(* IEC 61131-3 sources: RL_MAR/experiments/results/ablation/Ablation_no_post_process_deepseek-ai_DeepSeek-V3.2_20260602_235132 (part 3) *)

(* ---- med_69.st ---- *)
TYPE
    ST_ValueMapping : STRUCT
        valueInCondition : INT;
        valueOutResult : INT;
    END_STRUCT
END_TYPE

FUNCTION_BLOCK FB_ValueOut
VAR_INPUT
    valueIn : INT;
    conf : UINT;
END_VAR
VAR_OUTPUT
    ValueOut : INT;
END_VAR
VAR
    // Local variable for intermediate calculation
    tempResult : INT;
    // Array for conf=3 specific mappings
    conf3Mappings : ARRAY[1..3] OF ST_ValueMapping := [
        (valueInCondition := 0, valueOutResult := 0),
        (valueInCondition := 300, valueOutResult := 163),
        (valueInCondition := 600, valueOutResult := 331)
    ];
    // Array for conf=6/7 specific mapping
    conf67Mappings : ARRAY[1..1] OF ST_ValueMapping := [
        (valueInCondition := 100, valueOutResult := 319)
    ];
    i : INT;
    mappingFound : BOOL;
END_VAR

// Initialize output to 0
ValueOut := 0;

// Process based on configuration
CASE conf OF
    1, 2: // Divide valueIn by 10
        tempResult := valueIn / 10;
        // Ensure non-negative result
        IF tempResult >= 0 THEN
            ValueOut := tempResult;
        ELSE
            ValueOut := 0;
        END_IF;

    3: // Specific mappings for conf=3
        mappingFound := FALSE;
        FOR i := 1 TO 3 DO
            IF valueIn = conf3Mappings[i].valueInCondition THEN
                ValueOut := conf3Mappings[i].valueOutResult;
                mappingFound := TRUE;
                EXIT;
            END_IF;
        END_FOR;

        // If no mapping found, set to 0
        IF NOT mappingFound THEN
            ValueOut := 0;
        END_IF;

    6, 7: // Specific mapping for conf=6 or 7
        IF valueIn = conf67Mappings[1].valueInCondition THEN
            ValueOut := conf67Mappings[1].valueOutResult;
        ELSE
            ValueOut := 0;
        END_IF;

    ELSE // All other conf values (4,5,8,9,10, and any other)
        ValueOut := 0;
END_CASE;

// Final safety check to ensure non-negative output
IF ValueOut < 0 THEN
    ValueOut := 0;
END_IF;

END_FUNCTION_BLOCK;

(* ---- med_70.st ---- *)
FUNCTION_BLOCK EggIncubatorControl
VAR_INPUT
    StartButton : BOOL;          (* Rising edge triggers start *)
    StopButton : BOOL;           (* Rising edge triggers stop *)
    TemperatureSensor : REAL;    (* Current temperature in °C *)
    HumiditySensor : REAL;       (* Current humidity in % *)
END_VAR

VAR_OUTPUT
    HeatingElement : BOOL;       (* Controls heating element *)
    Humidifier : BOOL;           (* Controls humidifier *)
    EggTurningMotor : BOOL;      (* Controls turning motor *)
    IncubationInProgress : BOOL; (* Process status indicator *)
END_VAR

VAR
    TargetTemperature : REAL := 37.5;    (* Default target temperature *)
    TargetHumidity : REAL := 50.0;       (* Default target humidity *)
    TurnIntervalSeconds : INT := 3600;   (* Default turn interval *)
    TurnTimerSeconds : INT := 0;         (* Timer for turning cycle *)

    (* Edge detection for buttons *)
    StartButtonPrev : BOOL := FALSE;
    StopButtonPrev : BOOL := FALSE;
END_VAR

(* Edge detection for StartButton *)
IF StartButton AND NOT StartButtonPrev THEN
    (* Start condition: only if not already in progress *)
    IF NOT IncubationInProgress THEN
        IncubationInProgress := TRUE;
        TurnTimerSeconds := 0;
    END_IF;
END_IF;

(* Edge detection for StopButton *)
IF StopButton AND NOT StopButtonPrev THEN
    (* Immediate stop with reset *)
    IncubationInProgress := FALSE;
    HeatingElement := FALSE;
    Humidifier := FALSE;
    EggTurningMotor := FALSE;
    TurnTimerSeconds := 0;
END_IF;

(* Temperature control - only active when incubation is in progress *)
IF IncubationInProgress THEN
    HeatingElement := TemperatureSensor < TargetTemperature;
ELSE
    HeatingElement := FALSE;
END_IF;

(* Humidity control - only active when incubation is in progress *)
IF IncubationInProgress THEN
    Humidifier := HumiditySensor < TargetHumidity;
ELSE
    Humidifier := FALSE;
END_IF;

(* Egg turning cycle - only active when incubation is in progress *)
IF IncubationInProgress THEN
    (* Increment timer *)
    TurnTimerSeconds := TurnTimerSeconds + 1;

    (* Check if turn interval reached *)
    IF TurnTimerSeconds >= TurnIntervalSeconds THEN
        (* Toggle motor state *)
        EggTurningMotor := NOT EggTurningMotor;
        (* Reset timer *)
        TurnTimerSeconds := 0;
    END_IF;
ELSE
    (* Reset timer and motor when not in progress *)
    TurnTimerSeconds := 0;
    EggTurningMotor := FALSE;
END_IF;

(* Store previous button states for edge detection *)
StartButtonPrev := StartButton;
StopButtonPrev := StopButton;

END_FUNCTION_BLOCK

(* ---- med_71.st ---- *)
(*
    Fibonacci Calculator Function Block with Saturation Arithmetic
    Author: Senior PLC Commissioning Engineer
    Description: Calculates the N-th Fibonacci number with saturation at 32767
    Compliance: IEC 61131-3 Structured Text
*)

TYPE
    eFibonacciStatus : (
        eStatus_OK := 0,
        eStatus_Saturated := 1
    );
END_TYPE

FUNCTION_BLOCK FB_Fibonacci_Calculator
VAR_INPUT
    N : DINT := 5;  (* Target term index, 1-based *)
END_VAR
VAR_OUTPUT
    O : DINT := 1;  (* Calculated Fibonacci number *)
    Status : eFibonacciStatus := eStatus_OK;  (* Calculation status *)
END_VAR
VAR
    F1 : DINT := 1;  (* First previous term *)
    F2 : DINT := 1;  (* Second previous term *)
    Cnt : DINT := 2;  (* Current iteration counter *)
    Temp : DINT := 0;  (* Temporary variable for calculation *)
    MaxInt : DINT := 32767;  (* Maximum allowed value for saturation *)
END_VAR

(* Main calculation logic *)
IF N <= 0 THEN
    (* Invalid input - return 1 as specified for edge cases *)
    O := 1;
    Status := eStatus_OK;
ELSIF N <= 2 THEN
    (* Base cases: F(1) = 1, F(2) = 1 *)
    O := 1;
    Status := eStatus_OK;
ELSE
    (* Initialize for iterative calculation *)
    F1 := 1;
    F2 := 1;
    Cnt := 2;
    Status := eStatus_OK;

    (* Iterative calculation of Fibonacci numbers *)
    WHILE Cnt < N AND Status = eStatus_OK DO
        (* Check for potential overflow before calculation *)
        IF (F1 > MaxInt - F2) THEN
            (* Saturation condition detected *)
            O := MaxInt;
            Status := eStatus_Saturated;
        ELSE
            (* Calculate next Fibonacci number *)
            Temp := F1 + F2;

            (* Update previous terms for next iteration *)
            F1 := F2;
            F2 := Temp;

            (* Update counter *)
            Cnt := Cnt + 1;

            (* Set output to current term *)
            O := Temp;
        END_IF;
    END_WHILE;
END_IF;

END_FUNCTION_BLOCK;

(* ---- med_72.st ---- *)
FUNCTION_BLOCK DigitalSignageManagement
VAR_INPUT
    DisplayLocations : ARRAY[1..10] OF BOOL; (* TRUE = Display online, FALSE = Display offline *)
    ContentSource : ARRAY[1..10] OF INT; (* Desired content: 1=News, 2=Weather, 3=Promo, 0/other=None *)
END_VAR
VAR_OUTPUT
    CurrentContent : ARRAY[1..10] OF INT; (* Actual displayed content: 1=News, 2=Weather, 3=Promo, 0=None *)
END_VAR
VAR
    i : INT; (* Loop counter *)
END_VAR

(* Main processing loop: evaluates all 10 locations each scan cycle *)
FOR i := 1 TO 10 DO
    IF DisplayLocations[i] THEN
        (* Display is active: validate content code *)
        IF (ContentSource[i] = 1) OR (ContentSource[i] = 2) OR (ContentSource[i] = 3) THEN
            CurrentContent[i] := ContentSource[i]; (* Assign valid content *)
        ELSE
            CurrentContent[i] := 0; (* Invalid content code -> display nothing *)
        END_IF;
    ELSE
        (* Display is inactive: force no content *)
        CurrentContent[i] := 0;
    END_IF;
END_FOR;

END_FUNCTION_BLOCK

(* ---- med_73.st ---- *)
FUNCTION_BLOCK RoboticWeldingSystem
VAR_INPUT
    RobotArm1Ready : BOOL;    (* Input for robot arm 1 ready status *)
    RobotArm2Ready : BOOL;    (* Input for robot arm 2 ready status *)
    WeldingGunReady : BOOL;   (* Input for welding gun ready status *)
    StartButton : BOOL;       (* Input for start button press *)
    StopButton : BOOL;        (* Input for stop button press *)
END_VAR

VAR_OUTPUT
    WeldingTrigger : BOOL;    (* Output to trigger welding *)
    WeldingComplete : BOOL;   (* Output indicating welding completion *)
END_VAR

VAR
    bAllReady : BOOL;         (* Internal flag for all ready signals *)
    bStartCondition : BOOL;   (* Internal flag for valid start condition *)
END_VAR

(* Main logic for welding control *)
bAllReady := RobotArm1Ready AND RobotArm2Ready AND WeldingGunReady;
bStartCondition := bAllReady AND StartButton;

(* Priority: Stop button has highest precedence *)
IF StopButton THEN
    (* Safety stop: immediately halt welding and indicate completion *)
    WeldingTrigger := FALSE;
    WeldingComplete := TRUE;
ELSIF bStartCondition THEN
    (* Valid start condition: begin welding *)
    WeldingTrigger := TRUE;
    WeldingComplete := FALSE;
ELSE
    (* Default state: no welding, process complete *)
    WeldingTrigger := FALSE;
    WeldingComplete := TRUE;
END_IF;

END_FUNCTION_BLOCK

(* ---- med_74.st ---- *)
(*
    Traffic Light Control System
    FUNCTION_BLOCK: TrafficManagementSystem
    Description: Controls two independent pairs of traffic lights based on vehicle count comparison.
                 Handles equal counts by maintaining the last state.
    Author: Senior PLC Commissioning Engineer
    Standard: IEC 61131-3
*)

FUNCTION_BLOCK TrafficManagementSystem
VAR_INPUT
    (* Primary vehicle count inputs *)
    VehicleCount1 : INT; (* Vehicle count at intersection 1 *)
    VehicleCount2 : INT; (* Vehicle count at intersection 2 *)
    VehicleCount3 : INT; (* Vehicle count at intersection 3 *)
    VehicleCount4 : INT; (* Vehicle count at intersection 4 *)

    (* System control inputs - from agent 3uSa *)
    EmergencyOverride : BOOL := FALSE; (* Emergency override active *)
    ManualMode : BOOL := FALSE; (* Manual control mode active *)
    ManualGreen1 : BOOL := FALSE; (* Manual green for intersection 1 *)
    ManualGreen2 : BOOL := FALSE; (* Manual green for intersection 2 *)
    ManualGreen3 : BOOL := FALSE; (* Manual green for intersection 3 *)
    ManualGreen4 : BOOL := FALSE; (* Manual green for intersection 4 *)
    SystemReset : BOOL := FALSE; (* System reset command *)
    MinimumGreenTime : TIME := T#5s; (* Minimum green time duration *)
    YellowBlinkTimer : TIME := T#1s; (* Yellow blink interval *)
END_VAR

VAR_OUTPUT
    (* Primary traffic light outputs *)
    TrafficLight1 : BOOL; (* Green light for intersection 1 *)
    TrafficLight2 : BOOL; (* Green light for intersection 2 *)
    TrafficLight3 : BOOL; (* Green light for intersection 3 *)
    TrafficLight4 : BOOL; (* Green light for intersection 4 *)

    (* Additional outputs - from agent 3uSa *)
    YellowLight1 : BOOL; (* Yellow light for intersection 1 *)
    YellowLight2 : BOOL; (* Yellow light for intersection 2 *)
    YellowLight3 : BOOL; (* Yellow light for intersection 3 *)
    YellowLight4 : BOOL; (* Yellow light for intersection 4 *)
    SystemFault : BOOL; (* System fault indicator *)
    CurrentActivePair : INT; (* Currently active pair (1 or 2) *)
END_VAR

VAR
    (* Internal state variables *)
    LastState1 : BOOL := FALSE; (* Last state for pair 1 *)
    LastState3 : BOOL := FALSE; (* Last state for pair 2 *)

    (* Timer instances - from agent 3uSa *)
    GreenTimer1 : TON;
    GreenTimer2 : TON;
    GreenTimer3 : TON;
    GreenTimer4 : TON;
    YellowTimer1 : TON;
    YellowTimer2 : TON;
    YellowTimer3 : TON;
    YellowTimer4 : TON;
    BlinkTimer : TON;
    FaultTimer : TON;

    (* System status flags - from agent 3uSa *)
    ManualOverrideActive : BOOL := FALSE;
    EmergencyActive : BOOL := FALSE;
    SystemInitialized : BOOL := FALSE;
    FaultCondition : BOOL := FALSE;
    BlinkState : BOOL := FALSE;
    TransitionInProgress : BOOL := FALSE;

    (* Vehicle count tracking - from agent 3uSa *)
    LastVehicleCount1 : INT := 0;
    LastVehicleCount2 : INT := 0;
    LastVehicleCount3 : INT := 0;
    LastVehicleCount4 : INT := 0;
    VehicleCountDelta1 : INT := 0;
    VehicleCountDelta2 : INT := 0;
    VehicleCountDelta3 : INT := 0;
    VehicleCountDelta4 : INT := 0;

    (* Control variables *)
    Pair1Green : BOOL := FALSE;
    Pair2Green : BOOL := FALSE;
    EqualCountFlag : BOOL := FALSE;
    PriorityThreshold : INT := 5; (* Minimum difference to change state *)

    (* Temporary variables for logic *)
    tmpLight1 : BOOL;
    tmpLight2 : BOOL;
    tmpLight3 : BOOL;
    tmpLight4 : BOOL;
END_VAR

(* Main program logic *)
METHOD MainLogic : BOOL
VAR_INPUT
    countA : INT;
    countB : INT;
    lastState : BOOL;
END_VAR
VAR_OUTPUT
    result : BOOL;
END_VAR
    (* Core comparison logic with equal count handling *)
    IF countA > countB THEN
        result := TRUE;
    ELSIF countB > countA THEN
        result := FALSE;
    ELSE
        (* Equal counts - maintain last state *)
        result := lastState;
    END_IF;
END_METHOD

(* System initialization *)
IF SystemReset OR NOT SystemInitialized THEN
    (* Reset all states *)
    LastState1 := FALSE;
    LastState3 := FALSE;
    TrafficLight1 := FALSE;
    TrafficLight2 := FALSE;
    TrafficLight3 := FALSE;
    TrafficLight4 := FALSE;
    YellowLight1 := FALSE;
    YellowLight2 := FALSE;
    YellowLight3 := FALSE;
    YellowLight4 := FALSE;
    SystemFault := FALSE;
    CurrentActivePair := 0;
    SystemInitialized := TRUE;
    ManualOverrideActive := FALSE;
    EmergencyActive := FALSE;
    FaultCondition := FALSE;
    TransitionInProgress := FALSE;

    (* Reset timers *)
    GreenTimer1(IN:=FALSE);
    GreenTimer2(IN:=FALSE);
    GreenTimer3(IN:=FALSE);
    GreenTimer4(IN:=FALSE);
    YellowTimer1(IN:=FALSE);
    YellowTimer2(IN:=FALSE);
    YellowTimer3(IN:=FALSE);
    YellowTimer4(IN:=FALSE);
    BlinkTimer(IN:=FALSE);
    FaultTimer(IN:=FALSE);
END_IF;

(* Check for emergency override *)
EmergencyActive := EmergencyOverride;
ManualOverrideActive := ManualMode AND NOT EmergencyOverride;

(* Process vehicle count deltas *)
VehicleCountDelta1 := VehicleCount1 - LastVehicleCount1;
VehicleCountDelta2 := VehicleCount2 - LastVehicleCount2;
VehicleCountDelta3 := VehicleCount3 - LastVehicleCount3;
VehicleCountDelta4 := VehicleCount4 - LastVehicleCount4;

(* Update last vehicle counts *)
LastVehicleCount1 := VehicleCount1;
LastVehicleCount2 := VehicleCount2;
LastVehicleCount3 := VehicleCount3;
LastVehicleCount4 := VehicleCount4;

(* Main control logic *)
IF EmergencyActive THEN
    (* Emergency mode: all red *)
    tmpLight1 := FALSE;
    tmpLight2 := FALSE;
    tmpLight3 := FALSE;
    tmpLight4 := FALSE;
    YellowLight1 := FALSE;
    YellowLight2 := FALSE;
    YellowLight3 := FALSE;
    YellowLight4 := FALSE;
    CurrentActivePair := 0;

ELSIF ManualOverrideActive THEN
    (* Manual mode *)
    tmpLight1 := ManualGreen1;
    tmpLight2 := ManualGreen2;
    tmpLight3 := ManualGreen3;
    tmpLight4 := ManualGreen4;
    CurrentActivePair := 0;

    (* Ensure only one light per pair is green in manual mode *)
    IF ManualGreen1 AND ManualGreen2 THEN
        tmpLight1 := TRUE;
        tmpLight2 := FALSE;
    END_IF;
    IF ManualGreen3 AND ManualGreen4 THEN
        tmpLight3 := TRUE;
        tmpLight4 := FALSE;
    END_IF;

ELSE
    (* Automatic mode - apply core logic with equal count handling *)

    (* Process pair 1: Intersections 1 and 2 *)
    tmpLight1 := MainLogic(
        countA := VehicleCount1,
        countB := VehicleCount2,
        lastState := LastState1
    );
    tmpLight2 := NOT tmpLight1;

    (* Process pair 2: Intersections 3 and 4 *)
    tmpLight3 := MainLogic(
        countA := VehicleCount3,
        countB := VehicleCount4,
        lastState := LastState3
    );
    tmpLight4 := NOT tmpLight3;

    (* Update last states *)
    LastState1 := tmpLight1;
    LastState3 := tmpLight3;

    (* Set current active pair indicator *)
    IF tmpLight1 OR tmpLight2 THEN
        CurrentActivePair := 1;
    ELSIF tmpLight3 OR tmpLight4 THEN
        CurrentActivePair := 2;
    ELSE
        CurrentActivePair := 0;
    END_IF;

    (* Check for equal counts flag *)
    EqualCountFlag := (VehicleCount1 = VehicleCount2) OR (VehicleCount3 = VehicleCount4);
END_IF;

(* Apply minimum green time logic *)
(* Pair 1 *)
IF tmpLight1 THEN
    GreenTimer1(IN:=TRUE, PT:=MinimumGreenTime);
    IF NOT GreenTimer1.Q THEN
        tmpLight1 := FALSE;
        tmpLight2 := FALSE;
        YellowLight1 := TRUE;
    ELSE
        YellowLight1 := FALSE;
    END_IF;
ELSE
    GreenTimer1(IN:=FALSE);
    YellowLight1 := FALSE;
END_IF;

IF tmpLight2 THEN
    GreenTimer2(IN:=TRUE, PT:=MinimumGreenTime);
    IF NOT GreenTimer2.Q THEN
        tmpLight1 := FALSE;
        tmpLight2 := FALSE;
        YellowLight2 := TRUE;
    ELSE
        YellowLight2 := FALSE;
    END_IF;
ELSE
    GreenTimer2(IN:=FALSE);
    YellowLight2 := FALSE;
END_IF;

(* Pair 2 *)
IF tmpLight3 THEN
    GreenTimer3(IN:=TRUE, PT:=MinimumGreenTime);
    IF NOT GreenTimer3.Q THEN
        tmpLight3 := FALSE;
        tmpLight4 := FALSE;
        YellowLight3 := TRUE;
    ELSE
        YellowLight3 := FALSE;
    END_IF;
ELSE
    GreenTimer3(IN:=FALSE);
    YellowLight3 := FALSE;
END_IF;

IF tmpLight4 THEN
    GreenTimer4(IN:=TRUE, PT:=MinimumGreenTime);
    IF NOT GreenTimer4.Q THEN
        tmpLight3 := FALSE;
        tmpLight4 := FALSE;
        YellowLight4 := TRUE;
    ELSE
        YellowLight4 := FALSE;
    END_IF;
ELSE
    GreenTimer4(IN:=FALSE);
    YellowLight4 := FALSE;
END_IF;

(* Apply yellow blink timer *)
BlinkTimer(IN:=TRUE, PT:=YellowBlinkTimer);
IF BlinkTimer.Q THEN
    BlinkState := NOT BlinkState;
    BlinkTimer(IN:=FALSE);
END_IF;

(* Apply blinking to yellow lights *)
YellowLight1 := YellowLight1 AND BlinkState;
YellowLight2 := YellowLight2 AND BlinkState;
YellowLight3 := YellowLight3 AND BlinkState;
YellowLight4 := YellowLight4 AND BlinkState;

(* Final output assignment *)
TrafficLight1 := tmpLight1;
TrafficLight2 := tmpLight2;
TrafficLight3 := tmpLight3;
TrafficLight4 := tmpLight4;

(* Fault detection *)
FaultCondition := (VehicleCount1 < 0) OR (VehicleCount2 < 0) OR
                  (VehicleCount3 < 0) OR (VehicleCount4 < 0);

FaultTimer(IN:=FaultCondition, PT:=T#2s);
SystemFault := FaultTimer.Q;

END_FUNCTION_BLOCK;

(* ---- med_75.st ---- *)
(*
    Home Brewing System PLC Program
    FUNCTION_BLOCK: HomeBrewingSystem
    Description: Controls an automatic home brewing system with temperature control,
                 agitation based on water flow, and timed events for hops dispensing
                 and fermentation tank transfer.
    IEC 61131-3 Structured Text
*)

(* Custom Data Types *)
TYPE
    (* Process Stages Enumeration *)
    ProcessStage : (
        STAGE_IDLE := 0,
        STAGE_BREWING := 1,
        STAGE_HOPS_DISPENSED := 2,
        STAGE_FERMENTATION_READY := 3,
        STAGE_COMPLETE := 4
    );

    (* System Status Enumeration *)
    SystemStatus : (
        STATUS_DISABLED := 0,
        STATUS_READY := 1,
        STATUS_BREWING := 2,
        STATUS_ERROR := 3
    );

    (* Event Log Entry Structure *)
    EventLogEntry :
        STRUCT
            TimeStamp : TIME;
            EventCode : INT;
            Description : STRING(50);
        END_STRUCT;
END_TYPE

(*
    FUNCTION_BLOCK: HomeBrewingSystem
    Main control logic for the home brewing system
*)
FUNCTION_BLOCK HomeBrewingSystem
VAR_INPUT
    (* Primary Process Inputs *)
    TemperatureSensor : REAL;        (* Current temperature in °C *)
    WaterFlowSensor : REAL;          (* Current water flow in L/min *)
    BrewingStartTime : TIME;         (* Absolute start time of brewing process *)
    BrewingDuration : TIME;          (* Total brewing duration *)

    (* Configuration Parameters *)
    TemperatureSetpoint : REAL := 65.0;      (* Target brewing temperature *)
    FlowThreshold : REAL := 0.5;             (* Flow threshold for agitation *)
    HopsDispenseDelay : TIME := T#5h;        (* Time delay for hops dispensing *)
    FermentationDelay : TIME := T#48h;       (* Time delay for fermentation transfer *)
    TemperatureDeadband : REAL := 0.5;       (* Hysteresis for temperature control *)
    FlowDeadband : REAL := 0.1;              (* Hysteresis for flow control *)

    (* System Control Inputs *)
    SystemEnable : BOOL := TRUE;             (* Master enable for the system *)
    EmergencyStop : BOOL := FALSE;           (* Emergency stop input *)
    ManualHeatingOverride : BOOL := FALSE;   (* Manual heating control override *)
    ManualAgitationOverride : BOOL := FALSE; (* Manual agitation control override *)

    (* Calibration Offsets *)
    TemperatureCalibration : REAL := 0.0;    (* Temperature sensor calibration offset *)
    FlowCalibration : REAL := 0.0;           (* Flow sensor calibration offset *)
END_VAR

VAR_OUTPUT
    (* Primary Control Outputs *)
    HeatingElement : BOOL;           (* Control signal for heating element *)
    AgitationMotor : BOOL;           (* Control signal for agitation motor *)
    HopsDispenser : BOOL;            (* Control signal for hops dispenser *)
    FermentationTank : BOOL;         (* Control signal for fermentation tank transfer *)

    (* System Status Outputs *)
    SystemStatus : SystemStatus;     (* Current system status *)
    ProcessStage : ProcessStage;     (* Current process stage *)
    TemperatureAlarm : BOOL;         (* Temperature out of range alarm *)
    FlowAlarm : BOOL;                (* Flow out of range alarm *)

    (* Process Information *)
    ElapsedBrewingTime : TIME;       (* Time elapsed since brewing start *)
    TemperatureCorrected : REAL;      (* Calibrated temperature reading *)
    FlowCorrected : REAL;            (* Calibrated flow reading *)
    HopsDispenseReady : BOOL;        (* Indicates hops dispense is ready *)
    FermentationReady : BOOL;        (* Indicates fermentation transfer is ready *)
END_VAR

VAR
    (* Internal State Variables *)
    bHopsDispensed : BOOL := FALSE;          (* Flag to ensure single hops dispense *)
    bFermentationTriggered : BOOL := FALSE;  (* Flag to ensure single fermentation transfer *)
    bHeatingElementState : BOOL := FALSE;    (* Internal heating element state *)
    bAgitationMotorState : BOOL := FALSE;    (* Internal agitation motor state *)

    (* Process Timing Variables *)
    tCurrentTime : TIME;                     (* Current system time *)
    tElapsedTime : TIME;                     (* Elapsed brewing time *)
    tHopsDispenseTime : TIME;                (* Calculated hops dispense time *)
    tFermentationTime : TIME;                (* Calculated fermentation time *)

    (* Sensor Processing *)
    rTemperatureUpperLimit : REAL;           (* Upper temperature limit for deadband *)
    rTemperatureLowerLimit : REAL;           (* Lower temperature limit for deadband *)
    rFlowUpperThreshold : REAL;              (* Upper flow threshold for deadband *)
    rFlowLowerThreshold : REAL;              (* Lower flow threshold for deadband *)

    (* Safety and Interlocks *)
    bSafetyInterlock : BOOL := TRUE;         (* Safety interlock status *)
    bHeatingAllowed : BOOL := TRUE;          (* Heating permission flag *)
    bAgitationAllowed : BOOL := TRUE;        (* Agitation permission flag *)

    (* Event Logging *)
    aEventLog : ARRAY[1..50] OF EventLogEntry;  (* Circular buffer for event logging *)
    nLogIndex : INT := 1;                       (* Current log index *)

    (* Timers *)
    tmrHopsDispense : TON;                   (* Timer for hops dispense duration *)
    tmrFermentation : TON;                   (* Timer for fermentation transfer duration *)
END_VAR

(*
    Main Program Logic
*)

(* 1. Initialization and Safety Checks *)
(* Calculate deadband limits *)
rTemperatureUpperLimit := TemperatureSetpoint + (TemperatureDeadband / 2);
rTemperatureLowerLimit := TemperatureSetpoint - (TemperatureDeadband / 2);
rFlowUpperThreshold := FlowThreshold + (FlowDeadband / 2);
rFlowLowerThreshold := FlowThreshold - (FlowDeadband / 2);

(* Apply sensor calibration *)
TemperatureCorrected := TemperatureSensor + TemperatureCalibration;
FlowCorrected := WaterFlowSensor + FlowCalibration;

(* Get current system time *)
tCurrentTime := TIME();

(* Calculate elapsed brewing time *)
IF BrewingStartTime > T#0s THEN
    tElapsedTime := tCurrentTime - BrewingStartTime;

    (* Ensure elapsed time doesn't exceed brewing duration *)
    IF tElapsedTime > BrewingDuration THEN
        tElapsedTime := BrewingDuration;
    END_IF;
ELSE
    tElapsedTime := T#0s;
END_IF;

ElapsedBrewingTime := tElapsedTime;

(* Calculate event times *)
tHopsDispenseTime := HopsDispenseDelay;
tFermentationTime := FermentationDelay;

(* 2. Safety and System Status Management *)
(* Emergency stop handling *)
IF EmergencyStop THEN
    bSafetyInterlock := FALSE;
    SystemStatus := STATUS_ERROR;
ELSIF NOT SystemEnable THEN
    bSafetyInterlock := FALSE;
    SystemStatus := STATUS_DISABLED;
ELSE
    bSafetyInterlock := TRUE;

    (* Determine system status based on brewing state *)
    IF BrewingStartTime = T#0s THEN
        SystemStatus := STATUS_READY;
        ProcessStage := STAGE_IDLE;
    ELSIF tElapsedTime < BrewingDuration THEN
        SystemStatus := STATUS_BREWING;

        (* Update process stage *)
        IF tElapsedTime >= tFermentationTime THEN
            ProcessStage := STAGE_FERMENTATION_READY;
        ELSIF tElapsedTime >= tHopsDispenseTime THEN
            ProcessStage := STAGE_HOPS_DISPENSED;
        ELSE
            ProcessStage := STAGE_BREWING;
        END_IF;
    ELSE
        SystemStatus := STATUS_READY;
        ProcessStage := STAGE_COMPLETE;
    END_IF;
END_IF;

(* 3. Temperature Control Logic *)
(* Check temperature alarm condition *)
TemperatureAlarm := (TemperatureCorrected > (TemperatureSetpoint + 5.0)) OR
                    (TemperatureCorrected < (TemperatureSetpoint - 5.0));

(* Determine heating permission *)
bHeatingAllowed := bSafetyInterlock AND
                   (SystemStatus = STATUS_BREWING) AND
                   NOT TemperatureAlarm;

(* Temperature control with deadband *)
IF bHeatingAllowed THEN
    IF ManualHeatingOverride THEN
        bHeatingElementState := TRUE;
    ELSE
        (* Hysteresis control *)
        IF TemperatureCorrected < rTemperatureLowerLimit THEN
            bHeatingElementState := TRUE;
        ELSIF TemperatureCorrected > rTemperatureUpperLimit THEN
            bHeatingElementState := FALSE;
        END_IF;
        (* State persists between thresholds *)
    END_IF;
ELSE
    bHeatingElementState := FALSE;
END_IF;

(* 4. Flow Control Logic *)
(* Check flow alarm condition *)
FlowAlarm := (FlowCorrected > (FlowThreshold * 3.0)) OR
             (FlowCorrected < 0.0);

(* Determine agitation permission *)
bAgitationAllowed := bSafetyInterlock AND
                     (SystemStatus = STATUS_BREWING) AND
                     NOT FlowAlarm;

(* Flow control with deadband *)
IF bAgitationAllowed THEN
    IF ManualAgitationOverride THEN
        bAgitationMotorState := TRUE;
    ELSE
        (* Hysteresis control *)
        IF FlowCorrected > rFlowUpperThreshold THEN
            bAgitationMotorState := TRUE;
        ELSIF FlowCorrected < rFlowLowerThreshold THEN
            bAgitationMotorState := FALSE;
        END_IF;
        (* State persists between thresholds *)
    END_IF;
ELSE
    bAgitationMotorState := FALSE;
END_IF;

(* 5. Timed Event Control *)
(* Hops dispense control *)
IF (SystemStatus = STATUS_BREWING) AND
   (tElapsedTime >= tHopsDispenseTime) AND
   (NOT bHopsDispensed) THEN

    HopsDispenseReady := TRUE;

    (* Activate dispenser for 10 seconds *)
    tmrHopsDispense(IN := TRUE, PT := T#10s);

    IF tmrHopsDispense.Q THEN
        HopsDispenser := FALSE;
        bHopsDispensed := TRUE;
        tmrHopsDispense(IN := FALSE);
    ELSE
        HopsDispenser := TRUE;
    END_IF;
ELSE
    HopsDispenser := FALSE;
    HopsDispenseReady := FALSE;
    tmrHopsDispense(IN := FALSE);
END_IF;

(* Fermentation tank transfer control *)
IF (SystemStatus = STATUS_BREWING) AND
   (tElapsedTime >= tFermentationTime) AND
   (NOT bFermentationTriggered) THEN

    FermentationReady := TRUE;

    (* Activate transfer for 30 seconds *)
    tmrFermentation(IN := TRUE, PT := T#30s);

    IF tmrFermentation.Q THEN
        FermentationTank := FALSE;
        bFermentationTriggered := TRUE;
        tmrFermentation(IN := FALSE);
    ELSE
        FermentationTank := TRUE;
    END_IF;
ELSE
    FermentationTank := FALSE;
    FermentationReady := FALSE;
    tmrFermentation(IN := FALSE);
END_IF;

(* 6. Apply Safety Interlocks and Set Outputs *)
(* Apply final safety checks before setting outputs *)
IF bSafetyInterlock THEN
    HeatingElement := bHeatingElementState;
    AgitationMotor := bAgitationMotorState;

    (* Safety interlock: Prevent simultaneous heating and agitation *)
    IF bHeatingElementState AND bAgitationMotorState THEN
        AgitationMotor := FALSE;
    END_IF;

    (* Safety interlock: Prevent simultaneous hops dispense and fermentation transfer *)
    IF HopsDispenser AND FermentationTank THEN
        FermentationTank := FALSE;
    END_IF;
ELSE
    (* Emergency or disabled state - all outputs off *)
    HeatingElement := FALSE;
    AgitationMotor := FALSE;
    HopsDispenser := FALSE;
    FermentationTank := FALSE;
END_IF;

(* 7. Event Logging *)
(* Log significant state changes *)
IF (SystemStatus = STATUS_BREWING) AND (tElapsedTime = T#0s) THEN
    (* Log brewing start *)
    aEventLog[nLogIndex].TimeStamp := tCurrentTime;
    aEventLog[nLogIndex].EventCode := 100;
    aEventLog[nLogIndex].Description := 'Brewing process started';
    nLogIndex := nLogIndex MOD 50 + 1;
END_IF;

IF bHopsDispensed AND (HopsDispenser = FALSE) THEN
    (* Log hops dispensed *)
    aEventLog[nLogIndex].TimeStamp := tCurrentTime;
    aEventLog[nLogIndex].EventCode := 200;
    aEventLog[nLogIndex].Description := 'Hops dispensed';
    nLogIndex := nLogIndex MOD 50 + 1;
END_IF;

IF bFermentationTriggered AND (FermentationTank = FALSE) THEN
    (* Log fermentation transfer *)
    aEventLog[nLogIndex].TimeStamp := tCurrentTime;
    aEventLog[nLogIndex].EventCode := 300;
    aEventLog[nLogIndex].Description := 'Fermentation transfer completed';
    nLogIndex := nLogIndex MOD 50 + 1;
END_IF;

END_FUNCTION_BLOCK;

(* ---- med_76.st ---- *)
(*
    Multimedia Art Installation Control
    FUNCTION_BLOCK: MultimediaArtInstallationControl
    Description: Controls synchronization of audio, visual, and lighting elements
                 based on motion detection with safety protocols.
    State Machine: 0=IDLE, 1=ACTIVE, 2=SAFETY
*)

FUNCTION_BLOCK MultimediaArtInstallationControl
VAR_INPUT
    MotionSensor : BOOL;           (* Motion detection input *)
    AudioTrack : BOOL;             (* Selected audio track enable *)
    VisualContent : BOOL;          (* Selected visual content enable *)
    SystemCheck : BOOL;            (* Safety system check input *)
    PowerStatus : BOOL;            (* Power usage monitoring input *)
END_VAR

VAR_OUTPUT
    LightingControl : BOOL;        (* Lighting control output *)
    AudioControl : BOOL;           (* Audio playback control output *)
    VisualControl : BOOL;          (* Visual display control output *)
    TimerValue : INT;              (* Current activation timer value *)
    SystemStatus : BOOL;           (* Overall system status *)
END_VAR

VAR
    ActivationTimer : INT;         (* Timer for activation duration in seconds *)
    CurrentState : INT;            (* Current state identifier *)
    NextState : INT;               (* Next state identifier *)
    CycleCounter : INT;            (* Cycle counter for timing *)
    SafetyOverride : BOOL;         (* Safety override flag *)
    FirstCycle : BOOL := TRUE;     (* First cycle flag for initialization *)
END_VAR

VAR CONSTANT
    MAX_ACTIVATION_TIME : INT := 300;     (* 300 seconds maximum activation *)
    CYCLE_TIME_MS : INT := 100;           (* 100ms cycle time *)
    CYCLES_PER_SECOND : INT := 10;        (* 10 cycles per second for 100ms cycle *)
    STATE_IDLE : INT := 0;                (* Idle state identifier *)
    STATE_ACTIVE : INT := 1;              (* Active state identifier *)
    STATE_SAFETY : INT := 2;              (* Safety state identifier *)
END_VAR

(* Initialization on first cycle *)
IF FirstCycle THEN
    CurrentState := STATE_IDLE;
    NextState := STATE_IDLE;
    ActivationTimer := 0;
    CycleCounter := 0;
    SafetyOverride := FALSE;
    SystemStatus := TRUE;
    FirstCycle := FALSE;
END_IF;

(* Main state machine *)
CASE CurrentState OF
    STATE_IDLE:
        (* Actions executed in idle state *)
        LightingControl := FALSE;
        AudioControl := FALSE;
        VisualControl := FALSE;
        ActivationTimer := 0;
        CycleCounter := 0;
        TimerValue := 0;

        (* Transition logic from idle state *)
        IF NOT SystemCheck OR NOT PowerStatus THEN
            NextState := STATE_SAFETY;
        ELSIF MotionSensor AND SystemCheck AND PowerStatus THEN
            NextState := STATE_ACTIVE;
        ELSE
            NextState := STATE_IDLE;
        END_IF;

    STATE_ACTIVE:
        (* Actions executed in active state *)
        LightingControl := TRUE;
        AudioControl := AudioTrack AND SystemCheck;     (* Only activate if system check passes *)
        VisualControl := VisualContent AND SystemCheck; (* Only activate if system check passes *)

        (* Increment cycle counter for timing *)
        CycleCounter := CycleCounter + 1;

        (* Update timer every second (10 cycles at 100ms each) *)
        IF CycleCounter >= CYCLES_PER_SECOND THEN
            ActivationTimer := ActivationTimer + 1;
            CycleCounter := 0;
        END_IF;

        TimerValue := ActivationTimer;

        (* Transition logic from active state *)
        (* Safety override takes highest priority *)
        IF NOT SystemCheck OR NOT PowerStatus THEN
            NextState := STATE_SAFETY;
        (* Deactivate if no motion detected *)
        ELSIF NOT MotionSensor THEN
            NextState := STATE_IDLE;
        (* Deactivate if timer reaches maximum *)
        ELSIF ActivationTimer >= MAX_ACTIVATION_TIME THEN
            NextState := STATE_IDLE;
        (* Stay in active state *)
        ELSE
            NextState := STATE_ACTIVE;
        END_IF;

    STATE_SAFETY:
        (* Actions executed in safety state *)
        LightingControl := FALSE;
        AudioControl := FALSE;
        VisualControl := FALSE;
        ActivationTimer := 0;
        CycleCounter := 0;
        SystemStatus := FALSE;
        SafetyOverride := TRUE;

        (* Transition logic from safety state *)
        IF SystemCheck AND PowerStatus THEN
            SafetyOverride := FALSE;
            SystemStatus := TRUE;
            NextState := STATE_IDLE;
        ELSE
            NextState := STATE_SAFETY;
        END_IF;

END_CASE;

(* State transition *)
CurrentState := NextState;

(* Additional safety protocol: Power management consideration *)
IF LightingControl AND AudioControl AND VisualControl THEN
    (* Optional: Implement staggered activation or power limiting *)
    (* based on specific installation power requirements *)
END_IF;

END_FUNCTION_BLOCK

(* ---- med_77.st ---- *)
(*
    FUNCTION_BLOCK: OutdoorLEDLightingControl
    DESCRIPTION: Controls a modular outdoor LED lighting system based on ambient light, motion detection, and an energy-saving setting.
    LOGIC PRIORITY:
        1. Motion Detection Override: Lights ON if motion is detected.
        2. Ambient/Energy-Saving Logic: Lights ON only if ambient light < 50.0 AND energy-saving is OFF (when no motion is detected).
    OUTPUTS:
        Light: Controls the LED lights (TRUE = ON).
        EnergyMode: Reflects the current state of the EnergySaving input.
*)

FUNCTION_BLOCK OutdoorLEDLightingControl
VAR_INPUT
    AmbientLight : REAL;   (* Ambient light intensity in Lux *)
    MotionSensor : BOOL;   (* TRUE = Motion detected *)
    EnergySaving : BOOL;   (* TRUE = Energy saving mode is ON *)
END_VAR

VAR_OUTPUT
    Light      : BOOL;     (* Control output for the LED lights *)
    EnergyMode : BOOL;     (* Current energy-saving mode status *)
END_VAR

VAR
    // No internal variables required for this logic
END_VAR

// Main Control Logic
// 1. Energy Mode Status: Always reflect the input state.
EnergyMode := EnergySaving;

// 2. Light Control Logic
IF MotionSensor THEN
    // Motion Detection Override: Lights ON regardless of other conditions.
    Light := TRUE;
ELSE
    // No motion detected: Evaluate ambient light and energy-saving setting.
    IF (AmbientLight < 50.0) AND (NOT EnergySaving) THEN
        Light := TRUE;
    ELSE
        Light := FALSE;
    END_IF;
END_IF;

END_FUNCTION_BLOCK

(* ---- med_78.st ---- *)
FUNCTION_BLOCK RetractableRoofControl
VAR_INPUT
    RainSensor : BOOL;           (* TRUE when rain is detected *)
    WindSensor : BOOL;           (* TRUE when strong wind is detected *)
    TemperatureSensor : REAL;    (* Current temperature in degrees *)
END_VAR

VAR_OUTPUT
    RoofMotor : BOOL;            (* TRUE to close roof, FALSE to open roof *)
END_VAR

VAR
    CombinedCondition : BOOL;    (* Rain AND Wind condition *)
    RainOnlyCondition : BOOL;    (* Rain without strong wind *)
    LowTempCondition : BOOL;     (* Temperature below threshold *)
    TempThreshold : REAL := 20.0; (* Temperature threshold for closing roof *)
END_VAR

(* Evaluate conditions in order of priority *)
CombinedCondition := RainSensor AND WindSensor;
RainOnlyCondition := RainSensor AND NOT CombinedCondition;
LowTempCondition := (TemperatureSensor < TempThreshold) AND NOT CombinedCondition AND NOT RainOnlyCondition;

(* Apply control logic with strict priority *)
IF CombinedCondition THEN
    (* Highest priority: Both rain and strong wind detected *)
    RoofMotor := TRUE;
ELSIF RainOnlyCondition THEN
    (* Second priority: Rain detected without strong wind *)
    RoofMotor := TRUE;
ELSIF LowTempCondition THEN
    (* Third priority: Low temperature without rain or strong wind *)
    RoofMotor := TRUE;
ELSE
    (* Normal conditions: Open the roof *)
    RoofMotor := FALSE;
END_IF;

END_FUNCTION_BLOCK;

(* ---- med_79.st ---- *)
(* ================================================================ *)
(* CAPSULE FILLING MACHINE CONTROL FUNCTION BLOCK                   *)
(* IEC 61131-3 Structured Text                                     *)
(* Senior PLC Commissioning Engineer - Final Production Code       *)
(* ================================================================ *)

(* --- TYPE DEFINITIONS --- *)
TYPE
    (* State Machine Enumeration *)
    MachineState : (
        STATE_IDLE := 0,
        STATE_CONVEYING_IN := 1,
        STATE_FILLING := 2,
        STATE_CONVEYING_OUT := 3,
        STATE_ERROR := 4
    );
END_TYPE

(* --- FUNCTION BLOCK DEFINITION --- *)
FUNCTION_BLOCK CapsuleFillingMachineControl
VAR_INPUT
    (* Core Process Inputs *)
    CapsuleWeight : REAL;          (* Current capsule weight measurement *)
    TargetWeight : REAL;           (* Target weight to achieve *)
    CapsuleInPosition : BOOL;      (* TRUE when capsule is at filling station *)
    HopperEmpty : BOOL;            (* TRUE when hopper is completely empty *)

    (* Extended Inputs for Enhanced Control *)
    StartCycle : BOOL;             (* Rising edge triggers new cycle *)
    ResetErrors : BOOL;            (* Rising edge resets all errors *)
    EmergencyStop : BOOL;          (* Emergency stop input (TRUE = stop) *)

    (* Configuration Parameters *)
    WeightTolerance : REAL := 0.005;      (* Acceptable deviation from target *)
    MaxFillingTime : TIME := T#10S;       (* Maximum allowed filling duration *)
    MaxConveyingTime : TIME := T#3S;      (* Maximum conveying time *)
    ConveyingOutTime : TIME := T#1.5S;    (* Time to convey filled capsule out *)

    (* PID Controller Parameters *)
    Kp : REAL := 1.0;              (* Proportional gain *)
    Ti : TIME := T#2S;             (* Integral time *)
    Td : TIME := T#0.5S;           (* Derivative time *)
    PID_CycleTime : TIME := T#100MS; (* PID execution cycle *)
END_VAR

VAR_OUTPUT
    (* Primary Motor Controls *)
    FeederMotor : BOOL;            (* Controls material feed to hopper *)
    FillingMotor : BOOL;           (* Controls filling mechanism *)
    ConveyorMotor : BOOL;          (* Controls capsule conveyor *)
    FillingInProgress : BOOL;      (* TRUE during active filling *)

    (* Status and Diagnostic Outputs *)
    SystemReady : BOOL;            (* TRUE when system is ready for operation *)
    CycleComplete : BOOL;          (* TRUE when cycle completes successfully *)
    CurrentState : MachineState;   (* Current state machine state *)

    (* Error Flags *)
    CapsuleNotDetectedError : BOOL;    (* Capsule not detected in time *)
    FillingTimeoutError : BOOL;        (* Filling took too long *)
    OverweightError : BOOL;            (* Capsule already at/above target *)
    HopperEmptyError : BOOL;           (* Hopper is empty *)
    EmergencyStopActive : BOOL;        (* Emergency stop is active *)

    (* Process Monitoring *)
    PIDOutput : REAL;              (* Current PID controller output *)
    WeightDeviation : REAL;        (* Current deviation from target *)
    FillingTimeElapsed : TIME;     (* Time spent in filling state *)
END_VAR

VAR
    (* State Machine Variables *)
    CurrentStateInternal : MachineState := STATE_IDLE;
    PreviousState : MachineState;

    (* Timer Instances *)
    ConveyingTimer : TON;
    FillingTimer : TON;
    ConveyingOutTimer : TON;
    CapsuleDetectionTimer : TON;

    (* PID Controller *)
    PIDController : PID;
    PID_Enable : BOOL;
    ControlOutput : REAL;

    (* Process Flags *)
    CapsuleDetectedFlag : BOOL;
    FillingCompleteFlag : BOOL;
    ConveyingCompleteFlag : BOOL;
    ErrorResetFlag : BOOL;
    CycleStartFlag : BOOL;

    (* Error Latches *)
    CapsuleNotDetectedLatch : BOOL;
    FillingTimeoutLatch : BOOL;
    OverweightLatch : BOOL;
    HopperEmptyLatch : BOOL;
    EmergencyStopLatch : BOOL;

    (* Edge Detection *)
    StartCycleRisingEdge : R_TRIG;
    ResetErrorsRisingEdge : R_TRIG;

    (* Process Variables *)
    InitialWeightCheckPassed : BOOL;
    FillingMotorSpeed : REAL;
    ConveyorMotorSpeed : REAL;
    ActualFillingRate : REAL;
    CapsuleCount : DINT;
    ErrorCount : DINT;

    (* Internal Control Variables *)
    SafetyInterlock : BOOL;
    StateMachineEnabled : BOOL;
    ManualOverrideActive : BOOL;
END_VAR

(* ================================================================ *)
(* MAIN LOGIC - EXECUTED EVERY CYCLE                               *)
(* ================================================================ *)

(* --- Edge Detection for Control Signals --- *)
StartCycleRisingEdge(CLK := StartCycle);
ResetErrorsRisingEdge(CLK := ResetErrors);

(* --- Safety Interlock Calculation --- *)
SafetyInterlock := NOT HopperEmpty AND NOT EmergencyStop;
StateMachineEnabled := SafetyInterlock AND NOT ManualOverrideActive;

(* --- Error Reset Logic --- *)
IF ResetErrorsRisingEdge.Q THEN
    CapsuleNotDetectedLatch := FALSE;
    FillingTimeoutLatch := FALSE;
    OverweightLatch := FALSE;
    HopperEmptyLatch := FALSE;
    EmergencyStopLatch := FALSE;
    ErrorResetFlag := TRUE;
ELSE
    ErrorResetFlag := FALSE;
END_IF;

(* --- Emergency Stop Handling --- *)
IF EmergencyStop THEN
    EmergencyStopLatch := TRUE;
    CurrentStateInternal := STATE_IDLE;
END_IF;

(* --- Hopper Empty Error Latch --- *)
IF HopperEmpty THEN
    HopperEmptyLatch := TRUE;
END_IF;

(* --- System Ready Status --- *)
SystemReady := SafetyInterlock AND
               (CurrentStateInternal = STATE_IDLE) AND
               NOT EmergencyStopLatch AND
               NOT HopperEmptyLatch;

(* --- Cycle Start Flag --- *)
IF StartCycleRisingEdge.Q AND SystemReady THEN
    CycleStartFlag := TRUE;
ELSE
    CycleStartFlag := FALSE;
END_IF;

(* --- CRITICAL SAFETY CHECKS --- *)
(* 1. Hopper Empty Check - Immediate Safety Shutdown *)
IF HopperEmpty THEN
    FeederMotor := FALSE;
    FillingMotor := FALSE;
    ConveyorMotor := FALSE;
    FillingInProgress := FALSE;
    CycleComplete := FALSE;
    HopperEmptyError := TRUE;
    CurrentStateInternal := STATE_IDLE;
    RETURN;
END_IF;

(* 2. Emergency Stop Check *)
IF EmergencyStop THEN
    FeederMotor := FALSE;
    FillingMotor := FALSE;
    ConveyorMotor := FALSE;
    FillingInProgress := FALSE;
    CycleComplete := FALSE;
    EmergencyStopActive := TRUE;
    CurrentStateInternal := STATE_IDLE;
    RETURN;
END_IF;

(* 3. Initial Weight Validation *)
IF CapsuleWeight >= TargetWeight THEN
    FeederMotor := FALSE;
    FillingMotor := FALSE;
    ConveyorMotor := FALSE;
    FillingInProgress := FALSE;
    CycleComplete := FALSE;
    OverweightError := TRUE;
    OverweightLatch := TRUE;
    CurrentStateInternal := STATE_IDLE;
    RETURN;
END_IF;

(* --- STATE MACHINE EXECUTION --- *)
CASE CurrentStateInternal OF
    STATE_IDLE:
        (* Initialization and Waiting State *)
        FeederMotor := TRUE;                    (* Keep feeder running *)
        FillingMotor := FALSE;
        ConveyorMotor := FALSE;
        FillingInProgress := FALSE;
        CycleComplete := FALSE;
        PID_Enable := FALSE;

        (* Reset process flags *)
        CapsuleDetectedFlag := FALSE;
        FillingCompleteFlag := FALSE;
        ConveyingCompleteFlag := FALSE;

        (* Reset timers *)
        ConveyingTimer(IN := FALSE, PT := MaxConveyingTime);
        FillingTimer(IN := FALSE, PT := MaxFillingTime);
        ConveyingOutTimer(IN := FALSE, PT := ConveyingOutTime);
        CapsuleDetectionTimer(IN := FALSE, PT := MaxConveyingTime);

        (* Transition Conditions *)
        IF CycleStartFlag AND CapsuleInPosition THEN
            CapsuleDetectedFlag := TRUE;
            CurrentStateInternal := STATE_CONVEYING_IN;
        ELSIF CycleStartFlag THEN
            (* Start capsule detection timer *)
            CapsuleDetectionTimer(IN := TRUE, PT := MaxConveyingTime);
            CurrentStateInternal := STATE_CONVEYING_IN;
        END_IF;

    STATE_CONVEYING_IN:
        (* Move capsule to filling position *)
        ConveyorMotor := TRUE;
        FeederMotor := TRUE;
        FillingInProgress := FALSE;

        (* Start conveying timer *)
        ConveyingTimer(IN := TRUE, PT := MaxConveyingTime);

        (* Monitor for capsule detection *)
        IF CapsuleInPosition THEN
            CapsuleDetectedFlag := TRUE;
            CapsuleDetectionTimer(IN := FALSE, PT := MaxConveyingTime);
        END_IF;

        (* Transition Conditions *)
        IF CapsuleDetectedFlag THEN
            ConveyingTimer(IN := FALSE, PT := MaxConveyingTime);
            CurrentStateInternal := STATE_FILLING;
        ELSIF ConveyingTimer.Q THEN
            (* Timeout - capsule not detected *)
            CapsuleNotDetectedError := TRUE;
            CapsuleNotDetectedLatch := TRUE;
            CurrentStateInternal := STATE_ERROR;
        END_IF;

    STATE_FILLING:
        (* Precise Filling with PID Control *)
        ConveyorMotor := FALSE;
        FeederMotor := TRUE;
        FillingInProgress := TRUE;
        CycleComplete := FALSE;

        (* Enable PID Controller *)
        PID_Enable := TRUE;

        (* Configure and Execute PID *)
        PIDController.Kp := Kp;
        PIDController.Ti := Ti;
        PIDController.Td := Td;
        PIDController.Cycle := PID_CycleTime;

        PIDController.SP := TargetWeight;
        PIDController.PV := CapsuleWeight;
        PIDController.Enable := PID_Enable;
        PIDController.Execute();

        ControlOutput := PIDController.CO;
        PIDOutput := ControlOutput;

        (* Control Filling Motor based on PID output *)
        IF ControlOutput > 0.0 AND CapsuleWeight < TargetWeight THEN
            FillingMotor := TRUE;
            FillingMotorSpeed := ControlOutput;
        ELSE
            FillingMotor := FALSE;
            FillingMotorSpeed := 0.0;
        END_IF;

        (* Start filling timeout timer *)
        FillingTimer(IN := TRUE, PT := MaxFillingTime);
        FillingTimeElapsed := FillingTimer.ET;

        (* Calculate weight deviation *)
        WeightDeviation := TargetWeight - CapsuleWeight;

        (* Check for filling completion *)
        IF ABS(WeightDeviation) <= WeightTolerance THEN
            FillingCompleteFlag := TRUE;
            FillingMotor := FALSE;
            PID_Enable := FALSE;
            FillingTimer(IN := FALSE, PT := MaxFillingTime);
            CurrentStateInternal := STATE_CONVEYING_OUT;
        ELSIF FillingTimer.Q THEN
            (* Filling timeout error *)
            FillingTimeoutError := TRUE;
            FillingTimeoutLatch := TRUE;
            FillingMotor := FALSE;
            PID_Enable := FALSE;
            CurrentStateInternal := STATE_ERROR;
        END_IF;

    STATE_CONVEYING_OUT:
        (* Move filled capsule out of station *)
        FillingInProgress := FALSE;
        FillingMotor := FALSE;
        ConveyorMotor := TRUE;
        FeederMotor := TRUE;

        (* Start conveying out timer *)
        ConveyingOutTimer(IN := TRUE, PT := ConveyingOutTime);

        (* Transition Conditions *)
        IF ConveyingOutTimer.Q THEN
            ConveyorMotor := FALSE;
            CycleComplete := TRUE;
            CapsuleCount := CapsuleCount + 1;
            CurrentStateInternal := STATE_IDLE;
        END_IF;

    STATE_ERROR:
        (* Error State - All Motors Off *)
        FeederMotor := FALSE;
        FillingMotor := FALSE;
        ConveyorMotor := FALSE;
        FillingInProgress := FALSE;
        CycleComplete := FALSE;
        PID_Enable := FALSE;

        (* Reset timers *)
        ConveyingTimer(IN := FALSE, PT := MaxConveyingTime);
        FillingTimer(IN := FALSE, PT := MaxFillingTime);
        ConveyingOutTimer(IN := FALSE, PT := ConveyingOutTime);

        (* Wait for error reset *)
        IF ErrorResetFlag THEN
            CurrentStateInternal := STATE_IDLE;
        END_IF;

END_CASE;

(* --- Update Public State Output --- *)
CurrentState := CurrentStateInternal;

(* --- Update Previous State for Diagnostics --- *)
PreviousState := CurrentStateInternal;

(* --- Calculate Actual Filling Rate --- *)
IF FillingInProgress AND FillingTimeElapsed > T#0S THEN
    ActualFillingRate := CapsuleWeight / TIME_TO_REAL(FillingTimeElapsed);
ELSE
    ActualFillingRate := 0.0;
END_IF;

(* --- Update Error Count --- *)
ErrorCount := DINT_TO_DINT(CapsuleNotDetectedLatch) +
              DINT_TO_DINT(FillingTimeoutLatch) +
              DINT_TO_DINT(OverweightLatch) +
              DINT_TO_DINT(HopperEmptyLatch) +
              DINT_TO_DINT(EmergencyStopLatch);

END_FUNCTION_BLOCK

(* ---- med_80.st ---- *)
FUNCTION_BLOCK DoughMixerControl
VAR_INPUT
    IngredientsDetected : BOOL;
END_VAR

VAR_OUTPUT
    MixingInProgress : BOOL;
END_VAR

VAR
    MixingTimeElapsed : TIME;
    MixingTimeLimit : TIME := T#5S;
    IngredientsDetected_Prev : BOOL;
END_VAR

(* Rising edge detection for ingredient arrival *)
IF IngredientsDetected AND NOT IngredientsDetected_Prev THEN
    MixingInProgress := TRUE;
    MixingTimeElapsed := T#0S;
END_IF;

(* Stop conditions: ingredients removed OR time limit reached *)
IF NOT IngredientsDetected OR MixingTimeElapsed >= MixingTimeLimit THEN
    MixingInProgress := FALSE;
END_IF;

(* Timer increment only while mixing is active *)
IF MixingInProgress THEN
    MixingTimeElapsed := MixingTimeElapsed + T#1S;
END_IF;

(* Store previous state for edge detection *)
IngredientsDetected_Prev := IngredientsDetected;

END_FUNCTION_BLOCK;

(* ---- med_81.st ---- *)
FUNCTION_BLOCK SolarPanelTracking
VAR_INPUT
    CurrentTime : TIME;
    SolarIntensity : REAL;
END_VAR

VAR_OUTPUT
    PanelAngle : REAL;
END_VAR

VAR
    SunriseTime : TIME := T#6H;
    NoonTime : TIME := T#12H;
    SunsetTime : TIME := T#18H;
    MorningAngle : REAL := 30.0;
    NoonAngle : REAL := 60.0;
    EveningAngle : REAL := 30.0;
END_VAR

(* Main execution logic *)
IF SolarIntensity >= 90.0 THEN
    (* Solar intensity override - maximum energy capture *)
    PanelAngle := NoonAngle;
ELSE
    (* Time-based tracking logic *)
    IF (CurrentTime < SunriseTime) OR (CurrentTime >= SunsetTime) THEN
        (* Nighttime: panel horizontal *)
        PanelAngle := 0.0;
    ELSIF (CurrentTime >= SunriseTime) AND (CurrentTime < NoonTime) THEN
        (* Morning period *)
        PanelAngle := MorningAngle;
    ELSIF (CurrentTime >= NoonTime) AND (CurrentTime < SunsetTime) THEN
        (* Afternoon/Evening period *)
        PanelAngle := EveningAngle;
    ELSE
        (* Fallback safety condition *)
        PanelAngle := 0.0;
    END_IF;
END_IF;

END_FUNCTION_BLOCK;

(* ---- med_82.st ---- *)
FUNCTION_BLOCK PetFeederControl
VAR_INPUT
    CurrentTime : TIME; (* Current system time input *)
END_VAR
VAR_OUTPUT
    FoodDispense : BOOL; (* Food dispenser control signal *)
END_VAR
VAR
    FeedTime1 : TIME := T#8H0M0S; (* First feeding time - 8:00 AM *)
    FeedTime2 : TIME := T#12H0M0S; (* Second feeding time - 12:00 PM *)
    FeedTime3 : TIME := T#18H0M0S; (* Third feeding time - 6:00 PM *)
    FoodAmount : INT := 50; (* Amount of food to dispense in grams - currently unused *)
END_VAR

(* Main dispensing logic *)
FoodDispense := FALSE;

IF (CurrentTime >= FeedTime1) AND (CurrentTime < FeedTime1 + T#30S) THEN
    FoodDispense := TRUE;
ELSIF (CurrentTime >= FeedTime2) AND (CurrentTime < FeedTime2 + T#30S) THEN
    FoodDispense := TRUE;
ELSIF (CurrentTime >= FeedTime3) AND (CurrentTime < FeedTime3 + T#30S) THEN
    FoodDispense := TRUE;
END_IF;

END_FUNCTION_BLOCK

(* ---- med_83.st ---- *)
FUNCTION_BLOCK AmusementRideControl
VAR_INPUT
    StartButton : BOOL;    (* Start button input *)
    StopButton : BOOL;     (* Emergency stop button input *)
    SpeedSensor : REAL;    (* Speed sensor input (RPM) *)
    SafetySensor : BOOL;   (* Safety sensor status *)
END_VAR

VAR_OUTPUT
    MotorOn : BOOL := FALSE;    (* Motor control output *)
    BrakeOn : BOOL := TRUE;     (* Brake control output *)
END_VAR

VAR
    SpeedLimit : REAL := 60.0;  (* Maximum allowed speed in RPM *)
END_VAR

(* Main safety logic implementation *)
(* Emergency Stop has ABSOLUTE highest priority *)
IF StopButton THEN
    MotorOn := FALSE;
    BrakeOn := TRUE;

(* Normal operation monitoring when emergency stop is NOT active *)
ELSIF MotorOn THEN
    (* Continuous monitoring during operation *)
    IF (SpeedSensor > SpeedLimit) OR (NOT SafetySensor) THEN
        MotorOn := FALSE;
        BrakeOn := TRUE;
    END_IF;

(* Start condition evaluation *)
ELSIF StartButton AND (NOT StopButton) AND (SpeedSensor <= SpeedLimit) AND SafetySensor THEN
    MotorOn := TRUE;
    BrakeOn := FALSE;

(* Default fail-safe state *)
ELSE
    MotorOn := FALSE;
    BrakeOn := TRUE;
END_IF;

END_FUNCTION_BLOCK;

(* ---- med_85.st ---- *)
(* ============================================================================
   FINAL, PRODUCTION-READY FUNCTION_BLOCK FOR INDUSTRIAL SHREDDER CONTROL
   Senior PLC Commissioning Engineer Synthesis
   IEC 61131-3 Structured Text
   Priority: Safety > Normal Stop > Normal Start
   Features: Highest-priority emergency stop/jam, latching run command,
             fail-safe safety relay, manual reset after emergency.
============================================================================ *)

FUNCTION_BLOCK ShredderControl
VAR_INPUT
    (* Primary Command Inputs *)
    StartButton : BOOL;        (* Rising edge triggers start. Physical button. *)
    StopButton : BOOL;         (* Command to stop under normal conditions. *)
    EmergencyStop : BOOL;      (* TRUE = Emergency Stop Activated (Highest Priority). *)
    MaterialInFeed : BOOL;     (* TRUE = Material detected, requests auto-start. *)
    JammedSensor : BOOL;       (* TRUE = Jam detected (Highest Priority). *)
    (* System Feedback *)
    MotorStatus : BOOL;        (* Feedback contactor/motor running status. *)
    (* Safety & Reset *)
    ResetButton : BOOL;        (* Manual reset required after an emergency condition. *)
END_VAR

VAR_OUTPUT
    MotorControl : BOOL;       (* Command to motor contactor/ drive. *)
    SafetyRelay : BOOL;        (* Control for safety relay. TRUE = Safe, Energized. *)
    EmergencyLatched : BOOL;   (* TRUE indicates an emergency stop or jam is latched. *)
END_VAR

VAR
    (* State Variables *)
    MotorRunRequest : BOOL;    (* Internal latch for the run command. *)
    EmergencyCondition : BOOL; (* Combined emergency stop/jam signal. *)
    EmergencyLatch : BOOL;     (* Latch to remember an emergency occurred. *)
    StartPulse : BOOL;         (* Edge detection for StartButton. *)
    StartPulse_Memory : BOOL;  (* Memory for edge detection. *)
    ResetPulse : BOOL;         (* Edge detection for ResetButton. *)
    ResetPulse_Memory : BOOL;  (* Memory for edge detection. *)
END_VAR

(* ----------------------------------------------------------------------------
   INITIALIZATION & EDGE DETECTION
---------------------------------------------------------------------------- *)
(* Edge detection for push-button inputs (Start, Reset) *)
StartPulse := StartButton AND NOT StartPulse_Memory;
StartPulse_Memory := StartButton;

ResetPulse := ResetButton AND NOT ResetPulse_Memory;
ResetPulse_Memory := ResetButton;

(* ----------------------------------------------------------------------------
   SAFETY LOGIC: HIGHEST PRIORITY
---------------------------------------------------------------------------- *)
(* 1. Define the active emergency condition. *)
EmergencyCondition := EmergencyStop OR JammedSensor;

(* 2. Latch the emergency condition. Once TRUE, it stays TRUE until manually reset. *)
IF EmergencyCondition THEN
    EmergencyLatch := TRUE;
ELSIF ResetPulse THEN
    EmergencyLatch := FALSE;
END_IF;

(* ----------------------------------------------------------------------------
   MOTOR CONTROL LOGIC
---------------------------------------------------------------------------- *)
(* Priority 1: Emergency Latch (Highest Priority - Unconditional Stop) *)
IF EmergencyLatch THEN
    MotorRunRequest := FALSE;
(* Priority 2: Normal Stop Command *)
ELSIF StopButton THEN
    MotorRunRequest := FALSE;
(* Priority 3: Start Command (from button pulse OR material presence) *)
ELSIF StartPulse OR MaterialInFeed THEN
    MotorRunRequest := TRUE;
(* ELSE: Maintain current state (MotorRunRequest retains its value) *)
END_IF;

(* Final motor command is only valid if no active emergency condition exists. *)
MotorControl := MotorRunRequest AND NOT EmergencyCondition;

(* ----------------------------------------------------------------------------
   SAFETY RELAY LOGIC (FAIL-SAFE)
---------------------------------------------------------------------------- *)
(* Safety Relay is ONLY energized when:
   - No active emergency condition (EmergencyStop OR JammedSensor).
   - The emergency latch has been cleared (i.e., system has been reset).
   This ensures the relay drops out on any active fault and requires a reset. *)
SafetyRelay := NOT EmergencyCondition AND NOT EmergencyLatch;

(* ----------------------------------------------------------------------------
   STATUS OUTPUT
---------------------------------------------------------------------------- *)
EmergencyLatched := EmergencyLatch;

END_FUNCTION_BLOCK

(* ---- med_86.st ---- *)
FUNCTION_BLOCK FruitJuicingBottling
VAR_INPUT
    StartButton : BOOL;     (* Input for starting the process *)
    StopButton : BOOL;      (* Input for stopping the process *)
    FruitSelected : BOOL;   (* Input indicating fruit selection *)
END_VAR

VAR_OUTPUT
    JuiceProcessing : BOOL;     (* Output for controlling juice extraction *)
    BottleFilling : BOOL;       (* Output for controlling bottle filling *)
    CapPlacement : BOOL;        (* Output for placing caps on bottles *)
    Packaging : BOOL;           (* Output for packaging filled bottles *)
    ProcessInProgress : BOOL;   (* Indicator for an ongoing process *)
END_VAR

VAR
    bProcessRunning : BOOL;     (* Internal process state *)
    rTrigStart : R_TRIG;        (* Rising edge detection for StartButton *)
END_VAR

(* Rising edge detection for StartButton *)
rTrigStart(CLK := StartButton);

(* Process start/stop logic *)
IF rTrigStart.Q AND FruitSelected AND NOT bProcessRunning THEN
    bProcessRunning := TRUE;
END_IF;

IF StopButton OR NOT FruitSelected THEN
    bProcessRunning := FALSE;
END_IF;

(* Set outputs based on process state *)
ProcessInProgress := bProcessRunning;
JuiceProcessing := bProcessRunning;
BottleFilling := bProcessRunning;
CapPlacement := bProcessRunning;
Packaging := bProcessRunning;

END_FUNCTION_BLOCK

(* ---- med_87.st ---- *)
FUNCTION_BLOCK WaterDesalination
VAR_INPUT
    StartButton : BOOL;        (* Input for starting the desalination process *)
    StopButton : BOOL;         (* Input for stopping the desalination process *)
    SalinitySensor : REAL;     (* Input for salinity level measurement *)
END_VAR

VAR_OUTPUT
    SeawaterInletValve : BOOL;         (* Output for seawater inlet valve control *)
    FreshwaterOutletValve : BOOL;      (* Output for freshwater outlet valve control *)
    DesalinationInProgress : BOOL;     (* Indicator for an ongoing desalination process *)
END_VAR

VAR
    MaxSalinity : REAL := 35.0;        (* Maximum allowable salinity in ppm for freshwater *)
    SalinityControlSeconds : INT := 0; (* Timer for salinity control in seconds *)
    SalinityCheckTimer : TON;          (* IEC timer for 10-second interval *)
END_VAR

(* Timer for 10-second salinity check interval *)
SalinityCheckTimer(
    IN := DesalinationInProgress,
    PT := T#10S
);

(* Process Start/Stop Control *)
IF StopButton THEN
    (* Emergency/Manual Stop: Close valves, reset process *)
    DesalinationInProgress := FALSE;
    SeawaterInletValve := FALSE;
    FreshwaterOutletValve := FALSE;
    SalinityControlSeconds := 0;
ELSIF StartButton AND NOT DesalinationInProgress THEN
    (* Start Process: Open valves, set process active *)
    DesalinationInProgress := TRUE;
    SeawaterInletValve := TRUE;
    FreshwaterOutletValve := TRUE;
    SalinityControlSeconds := 0;
END_IF;

(* Salinity Monitoring and Control *)
IF DesalinationInProgress THEN
    (* Update timer display value (seconds) *)
    SalinityControlSeconds := TIME_TO_INT(SalinityCheckTimer.ET) / 1000;

    (* Check salinity every 10 seconds *)
    IF SalinityCheckTimer.Q THEN
        IF SalinitySensor > MaxSalinity THEN
            FreshwaterOutletValve := FALSE;    (* Close valve if salinity too high *)
        ELSE
            FreshwaterOutletValve := TRUE;     (* Keep valve open if salinity OK *)
        END_IF;

        (* Reset timer for next 10-second interval *)
        SalinityCheckTimer(IN := FALSE);
        SalinityCheckTimer(IN := TRUE);
    END_IF;
ELSE
    (* Process not active: Ensure valves are closed *)
    SeawaterInletValve := FALSE;
    FreshwaterOutletValve := FALSE;
END_IF;

END_FUNCTION_BLOCK

(* ---- med_88.st ---- *)
TYPE
    LockerStatusType : ARRAY[1..10] OF BOOL;
    LockerAccessCodeType : ARRAY[1..10] OF INT;
END_TYPE

FUNCTION_BLOCK SmartLockerControl
VAR_INPUT
    AccessCode : INT;     (* User entered access code *)
    LockerNumber : INT;   (* Selected locker number (1-10) *)
END_VAR
VAR_OUTPUT
    LockerOpen : BOOL;    (* TRUE when locker should open *)
END_VAR
VAR
    LockerStatus : LockerStatusType := [TRUE, TRUE, TRUE, TRUE, TRUE, TRUE, TRUE, TRUE, TRUE, TRUE];
    LockerAccessCode : LockerAccessCodeType := [1234, 5678, 9876, 4321, 6543, 7890, 3456, 8765, 2345, 6789];
    validLockerNumber : BOOL;
    codeMatches : BOOL;
END_VAR

(* Validate locker number is within range *)
validLockerNumber := (LockerNumber >= 1) AND (LockerNumber <= 10);

(* Check if access code matches for the specified locker *)
IF validLockerNumber THEN
    codeMatches := (AccessCode = LockerAccessCode[LockerNumber]);
ELSE
    codeMatches := FALSE;
END_IF;

(* Main access control logic *)
IF validLockerNumber AND codeMatches AND LockerStatus[LockerNumber] THEN
    LockerOpen := TRUE;
    LockerStatus[LockerNumber] := FALSE;  (* Mark locker as empty after opening *)
ELSE
    LockerOpen := FALSE;
END_IF;

END_FUNCTION_BLOCK;

(* ---- med_89.st ---- *)
FUNCTION_BLOCK SoilTestingDeviceControl
VAR_INPUT
    StartButton : BOOL; (* Input for starting the testing process *)
    SoilSampleDetected : BOOL; (* Input for detecting soil sample *)
END_VAR
VAR_OUTPUT
    NutrientPump : BOOL; (* Output to control nutrient pump *)
    pHAdjustmentPump : BOOL; (* Output to control pH adjustment pump *)
END_VAR
VAR
    pHSensorValue : REAL; (* Simulated pH sensor value *)
    NutrientSensorValue : REAL; (* Simulated nutrient sensor value *)
    TestingStatus : INT; (* Status: 0=Idle, 1=Testing, 2=Completed *)
    NutrientThreshold : REAL := 0.7; (* Nutrient level threshold for analysis *)
    pHThreshold : REAL := 6.5; (* pH level threshold for analysis *)
    tSampleVerification : TON; (* Timer for sample verification delay *)
    bStartButtonPrev : BOOL; (* Edge detection for StartButton *)
    bSampleDetectedPrev : BOOL; (* Edge detection for SoilSampleDetected *)
END_VAR

(* State Machine Implementation *)
CASE TestingStatus OF
    0: (* Idle State *)
        (* Initialize sensor values *)
        pHSensorValue := 7.0;
        NutrientSensorValue := 0.5;

        (* Ensure pumps are deactivated *)
        NutrientPump := FALSE;
        pHAdjustmentPump := FALSE;

        (* Reset verification timer *)
        tSampleVerification(IN:=FALSE, PT:=T#2S);

        (* Detect rising edge of StartButton to transition to Testing state *)
        IF StartButton AND NOT bStartButtonPrev THEN
            TestingStatus := 1;
            (* Activate pumps upon transition *)
            NutrientPump := TRUE;
            pHAdjustmentPump := TRUE;
        END_IF;

        (* Store current button state for next cycle *)
        bStartButtonPrev := StartButton;

    1: (* Testing State *)
        (* Update sensor values with limits *)
        NutrientSensorValue := REAL_MIN(NutrientSensorValue + 0.1, 0.9);
        pHSensorValue := REAL_MAX(pHSensorValue - 0.5, 4.0);

        (* Detect rising edge of SoilSampleDetected *)
        IF SoilSampleDetected AND NOT bSampleDetectedPrev THEN
            (* Start verification timer *)
            tSampleVerification(IN:=TRUE, PT:=T#2S);
        END_IF;

        (* Check for completion conditions after verification delay *)
        IF tSampleVerification.Q THEN
            IF (NutrientSensorValue >= NutrientThreshold) AND (pHSensorValue <= pHThreshold) THEN
                (* Conditions met - transition to Completed *)
                TestingStatus := 2;
                NutrientPump := FALSE;
                pHAdjustmentPump := FALSE;
            ELSE
                (* Conditions not met - reset timer for next detection *)
                tSampleVerification(IN:=FALSE);
            END_IF;
        END_IF;

        (* Store current sample detection state for next cycle *)
        bSampleDetectedPrev := SoilSampleDetected;

    2: (* Completed State *)
        (* Ensure pumps remain deactivated *)
        NutrientPump := FALSE;
        pHAdjustmentPump := FALSE;

        (* Reset timer *)
        tSampleVerification(IN:=FALSE, PT:=T#2S);

        (* Reset to Idle when StartButton is released *)
        IF NOT StartButton THEN
            TestingStatus := 0;
        END_IF;

END_CASE;

END_FUNCTION_BLOCK

(* ---- med_90.st ---- *)
(*
    FUNCTION_BLOCK: SushiConveyorControl
    Description: Controls an automated sushi conveyor belt with emergency stop, start/stop, and simulated rotation via timed on/off cycles.
    Priority: Emergency Stop (highest) > Start/Stop Control > Simulated Rotation.
    Note: This implementation uses a simple integer counter (ConveyorTimer) for timing. In a real PLC, this would typically be replaced by a hardware timer (TON) or a time-based increment.
*)

FUNCTION_BLOCK SushiConveyorControl
VAR_INPUT
    StartButton : BOOL;     (* Momentary input to start the conveyor *)
    StopButton : BOOL;      (* Momentary input to stop the conveyor *)
    EmergencyStop : BOOL;   (* Hardwired emergency stop signal *)
END_VAR

VAR_OUTPUT
    ConveyorMotor : BOOL;   (* Output signal to the conveyor motor contactor *)
END_VAR

VAR
    BeltRunning : BOOL;     (* Internal state: TRUE when conveyor is running *)
    ConveyorTimer : INT;    (* Counter for simulated rotation timing *)
    RotationTime : INT := 5; (* Duration of one motor ON cycle (e.g., seconds) *)
    CycleActive : BOOL;     (* Internal flag: TRUE during the ON part of the cycle *)
END_VAR

(* Main Logic Execution *)
BEGIN
    (* 1. EMERGENCY STOP - HIGHEST PRIORITY *)
    IF EmergencyStop THEN
        ConveyorMotor := FALSE;
        BeltRunning := FALSE;
        ConveyorTimer := 0;
        CycleActive := FALSE;
        RETURN; (* Immediate exit from the function block *)
    END_IF;

    (* 2. START/STOP CONTROL *)
    IF StartButton AND NOT BeltRunning THEN
        BeltRunning := TRUE;
        ConveyorTimer := 0;
        CycleActive := TRUE;
    ELSIF StopButton AND BeltRunning THEN
        BeltRunning := FALSE;
        ConveyorTimer := 0;
        CycleActive := FALSE;
        ConveyorMotor := FALSE;
    END_IF;

    (* 3. SIMULATED ROTATION (Timed On/Off Cycle) *)
    IF BeltRunning THEN
        (* Increment the timer to simulate passage of time *)
        ConveyorTimer := ConveyorTimer + 1;

        (* Check if the ON cycle duration has been reached *)
        IF ConveyorTimer >= RotationTime THEN
            ConveyorTimer := 0;       (* Reset timer for next cycle *)
            CycleActive := NOT CycleActive; (* Toggle between ON and OFF parts of the cycle *)
        END_IF;

        (* Motor is only energized during the active part of the cycle *)
        ConveyorMotor := CycleActive;
    ELSE
        (* Conveyor is not running, ensure motor is off and timer is reset *)
        ConveyorTimer := 0;
        CycleActive := FALSE;
        ConveyorMotor := FALSE;
    END_IF;

END_FUNCTION_BLOCK

(* ---- med_91.st ---- *)
TYPE AGV_Status :
STRUCT
    IsReady : BOOL;
    CurrentTask : INT;
    Position : INT;
    IsWorking : BOOL;
END_STRUCT
END_TYPE

FUNCTION_BLOCK AGVControlSystem
VAR_INPUT
    MaterialRequest : INT; (* New material request, valid if > 0 *)
    ExecuteCycle : BOOL := TRUE; (* Enable processing for the scan cycle *)
END_VAR
VAR_OUTPUT
    AGV1_Ready : BOOL := TRUE;
    AGV2_Ready : BOOL := TRUE;
    AGV3_Ready : BOOL := TRUE;
    QueueCount : INT := 0; (* Number of pending tasks *)
    SystemIdle : BOOL := TRUE; (* All AGVs ready AND queue empty *)
    ErrorCode : INT := 0; (* 0: OK, 1: Queue Overflow, 2: Invalid Request *)
END_VAR
VAR
    MaterialQueue : ARRAY[1..10] OF INT; (* FIFO queue for tasks *)
    QueueHead : INT := 1; (* Index of the next task to dequeue *)
    QueueTail : INT := 1; (* Index where the next task will be enqueued *)
    AGVs : ARRAY[1..3] OF AGV_Status := [(IsReady:=TRUE, CurrentTask:=0, Position:=0, IsWorking:=FALSE),
                                         (IsReady:=TRUE, CurrentTask:=0, Position:=0, IsWorking:=FALSE),
                                         (IsReady:=TRUE, CurrentTask:=0, Position:=0, IsWorking:=FALSE)];
    TaskAssignedThisCycle : BOOL; (* Prevents multiple assignments in one scan *)
    i : INT;
END_VAR

(* 1. Process new material request with validation and overflow protection *)
ErrorCode := 0;
IF ExecuteCycle THEN
    IF MaterialRequest > 0 THEN
        IF QueueCount < 10 THEN
            MaterialQueue[QueueTail] := MaterialRequest;
            QueueTail := QueueTail + 1;
            IF QueueTail > 10 THEN
                QueueTail := 1;
            END_IF;
            QueueCount := QueueCount + 1;
        ELSE
            ErrorCode := 1; (* Queue Overflow *)
        END_IF;
    ELSIF MaterialRequest < 0 THEN
        ErrorCode := 2; (* Invalid Request *)
    END_IF;

    (* 2. Priority-based task assignment (AGV1 > AGV2 > AGV3) *)
    TaskAssignedThisCycle := FALSE;
    FOR i := 1 TO 3 DO
        IF (AGVs[i].IsReady) AND (QueueCount > 0) AND (NOT TaskAssignedThisCycle) THEN
            AGVs[i].CurrentTask := MaterialQueue[QueueHead];
            AGVs[i].IsReady := FALSE;
            AGVs[i].IsWorking := TRUE;
            AGVs[i].Position := 0; (* Reset position at task start *)
            QueueHead := QueueHead + 1;
            IF QueueHead > 10 THEN
                QueueHead := 1;
            END_IF;
            QueueCount := QueueCount - 1;
            TaskAssignedThisCycle := TRUE;
        END_IF;
    END_FOR;

    (* 3. Simulate task execution and handle completion *)
    FOR i := 1 TO 3 DO
        IF AGVs[i].IsWorking THEN
            (* Simulate position update during task execution *)
            AGVs[i].Position := AGVs[i].Position + 1;

            (* Safety constraint: ensure non-negative position *)
            IF AGVs[i].Position < 0 THEN
                AGVs[i].Position := 0;
            END_IF;

            (* Task completion check - example: task completes after 10 position units *)
            IF AGVs[i].Position >= 10 THEN
                (* Release AGV resource *)
                AGVs[i].Position := 0;
                AGVs[i].CurrentTask := 0;
                AGVs[i].IsWorking := FALSE;
                AGVs[i].IsReady := TRUE;
            END_IF;
        END_IF;
    END_FOR;

    (* 4. Update output status *)
    AGV1_Ready := AGVs[1].IsReady;
    AGV2_Ready := AGVs[2].IsReady;
    AGV3_Ready := AGVs[3].IsReady;

    (* 5. State monitoring and synchronization *)
    SystemIdle := (QueueCount = 0) AND AGVs[1].IsReady AND AGVs[2].IsReady AND AGVs[3].IsReady;

    (* 6. Sanity checks for queue indices (defensive programming) *)
    IF QueueHead < 1 OR QueueHead > 10 THEN
        QueueHead := 1;
    END_IF;
    IF QueueTail < 1 OR QueueTail > 10 THEN
        QueueTail := 1;
    END_IF;
    IF QueueCount < 0 THEN
        QueueCount := 0;
    ELSIF QueueCount > 10 THEN
        QueueCount := 10;
    END_IF;
END_IF;

END_FUNCTION_BLOCK

(* ---- med_84.st ---- *)
(* ======================================================================
   Parcel Sorting System - FUNCTION_BLOCK
   ======================================================================
   Description: Controls a conveyor belt and two sorting gates to route
                parcels based on size and destination code.
   Inputs:  ParcelSizeSensor - REAL value representing parcel size
            DestinationCodeSensor - INT code (1=Location A, 2=Location B)
   Outputs: ConveyorBeltMotor - BOOL motor control (TRUE=On)
            SortingGate1 - BOOL gate control (TRUE=Open)
            SortingGate2 - BOOL gate control (TRUE=Open)
   Sorting Logic:
     - Large parcels (Size ≥ LARGE_SIZE_THRESHOLD) → Sorting Gate 1
     - Small parcels to Location A (Dest=1) → Sorting Gate 2
     - Small parcels to Location B (Dest=2) → No gate activation
     - Invalid inputs → Stop conveyor, close both gates
   ====================================================================== *)

(* ----------------------------------------------------------------------
   Constants and Configuration Parameters
   ---------------------------------------------------------------------- *)
VAR CONSTANT
    LARGE_SIZE_THRESHOLD : REAL := 50.0;  (* Size threshold for large parcels *)
    MIN_VALID_SIZE : REAL := 0.001;       (* Minimum valid parcel size *)
END_VAR

(* ----------------------------------------------------------------------
   Internal Variables for State Management
   ---------------------------------------------------------------------- *)
VAR
    (* State flags *)
    bInputsValid : BOOL;      (* TRUE when both sensor inputs are valid *)
    bIsLargeParcel : BOOL;    (* TRUE when parcel size ≥ threshold *)
    bDestIsA : BOOL;          (* TRUE when destination code = 1 (Location A) *)
    bDestIsB : BOOL;          (* TRUE when destination code = 2 (Location B) *)

    (* Intermediate calculation variables *)
    rParcelSize : REAL;       (* Local copy of size input *)
    iDestCode : INT;          (* Local copy of destination input *)
END_VAR

(* ======================================================================
   FUNCTION_BODY: Main Control Logic
   ====================================================================== *)

(* ----------------------------------------------------------------------
   STEP 1: Read and Validate Inputs
   ---------------------------------------------------------------------- *)
(* Make local copies of inputs for processing *)
rParcelSize := ParcelSizeSensor;
iDestCode := DestinationCodeSensor;

(* Validate parcel size: must be positive and above minimum threshold *)
IF rParcelSize >= MIN_VALID_SIZE THEN
    (* Validate destination code: must be 1 or 2 *)
    IF (iDestCode = 1) OR (iDestCode = 2) THEN
        bInputsValid := TRUE;
    ELSE
        bInputsValid := FALSE;
    END_IF;
ELSE
    bInputsValid := FALSE;
END_IF;

(* ----------------------------------------------------------------------
   STEP 2: Process Valid Inputs - Determine Parcel Characteristics
   ---------------------------------------------------------------------- *)
IF bInputsValid THEN
    (* Determine if parcel is large based on threshold *)
    IF rParcelSize >= LARGE_SIZE_THRESHOLD THEN
        bIsLargeParcel := TRUE;
    ELSE
        bIsLargeParcel := FALSE;
    END_IF;

    (* Determine destination *)
    bDestIsA := (iDestCode = 1);
    bDestIsB := (iDestCode = 2);

    (* ------------------------------------------------------------------
       STEP 3: Apply Sorting Rules (Decision Matrix)
       ------------------------------------------------------------------ *)

    (* Rule 1: Conveyor runs for all valid inputs *)
    ConveyorBeltMotor := TRUE;

    (* Rule 2: Large parcels go to Gate 1 (regardless of destination) *)
    IF bIsLargeParcel THEN
        SortingGate1 := TRUE;
        SortingGate2 := FALSE;
    (* Rule 3: Small parcels to Location A go to Gate 2 *)
    ELSIF bDestIsA THEN
        SortingGate1 := FALSE;
        SortingGate2 := TRUE;
    (* Rule 4: Small parcels to Location B - no gate activation *)
    ELSIF bDestIsB THEN
        SortingGate1 := FALSE;
        SortingGate2 := FALSE;
    (* Fallback: Should not occur if inputs are valid, but for safety *)
    ELSE
        SortingGate1 := FALSE;
        SortingGate2 := FALSE;
    END_IF;

(* ----------------------------------------------------------------------
   STEP 4: Handle Invalid Inputs - Error State
   ---------------------------------------------------------------------- *)
ELSE
    (* Invalid inputs: Stop conveyor and close both gates *)
    ConveyorBeltMotor := FALSE;
    SortingGate1 := FALSE;
    SortingGate2 := FALSE;

    (* Reset internal state variables for safety *)
    bIsLargeParcel := FALSE;
    bDestIsA := FALSE;
    bDestIsB := FALSE;
END_IF;

(* ======================================================================
   END OF FUNCTION_BODY
   ====================================================================== *)
